{attribute 'qualified_only'}
{attribute 'strict'}
TYPE E_Cmd :
( 	
	INITIALISE:=0,
	AlarmReset,
	ColumnAlarmReset,
	TIUSlideIn,
	TIUSlideOut,
	TIUDrawerUp,
	TIUDrawerDown,
	TIUSlideOutRetry,
	TIUSlideOutCancel,
	DPSPowerON,
	DPSPowerOFF,
	DPSPowerAuto,
	AP240ACPowerON,
	AP240ACPowerOFF,
	APAirValveON,
	APAirValveOFF,
	TstAirValveON,
	TstAirValveOFF,
	CellDoorOpen,
	CellDoorClose,
	CancelBuffer,
	SetLEDON,
	SetLEDOFF, 
	SetLEDBlink,
	DCCellFrontDoorOpen,
	DCCellFrontDoorClose,
	TIUSocketAirOn_1,
	TIUSocketAirOn_2,
	TIUSocketAirOff_1,
	TIUSocketAirOff_2,
	EnableTester,
	DisableTester,
	EnableTCU,
	DisableTCU,
	EnableTII,
	DisableTII,
	SetTCUSafeState,
	SetSolenoidValvesON,
	SetSolenoidValvesOFF,
	Secondary24VPowerON,
	Secondary24VPowerOFF
);
END_TYPE

(* stored: Version 1.1.0.1, ProductVersion 3.1.4022.18
   EnumerationTextList E_Cmd: Id {ac96e949-a18f-4c77-a16f-32c06176c4b3} *)
